// TwinCAT 3 PLC project Lab1
// ProgramVersion: 3.1.4023.0
// libraries:
//   Tc2_Standard, * (Beckhoff Automation GmbH)
//   Tc2_System, * (Beckhoff Automation GmbH)
//   Tc3_Module, * (Beckhoff Automation GmbH)
//   VisuDialogs, * (System)
// project tree:
//   DUTs/ E_CraneMode.TcDUT, E_CraneStatus.TcDUT, ST_pPistonRange.TcDUT
//   / GlobalTextList.TcGTLO, PlcTask.TcTTO (not stored), Visualization Manager.TcVMO (not stored)
//   GVLs/ HMI.TcGVL, Inputs.TcGVL, Outputs.TcGVL, Parameters.TcGVL
//   POUs/ CraneSimulation.TcPOU, F_BarToEng.TcPOU, F_LminToEng.TcPOU, F_UpdateParametersByReference.TcPOU, MAIN.TcPOU
//   VISUs/ CraneHMI.TcVIS

// ---- DUTs/E_CraneMode.TcDUT
{attribute 'qualified_only'}
{attribute 'strict'}
TYPE E_CraneMode :
(
	Manual,
	Auto
);
END_TYPE

// ---- DUTs/E_CraneStatus.TcDUT
{attribute 'qualified_only'}
{attribute 'strict'}
TYPE E_CraneStatus :
(
	Ready,
	Starting,
	Running,
	Faulty
);
END_TYPE

// ---- DUTs/ST_pPistonRange.TcDUT
TYPE ST_pPistonRange :
STRUCT
	fPistonPosMin : LREAL := 0.0;
	fPistonPosMax : LREAL := 0.5;
END_STRUCT
END_TYPE

// ---- GVLs/HMI.TcGVL
{attribute 'qualified_only'}
VAR_GLOBAL
	sPistonEndStopMessages : STRING;
END_VAR

// ---- GVLs/Inputs.TcGVL
{attribute 'qualified_only'}
VAR_GLOBAL
	bEnableSimulation : BOOL; 
	bStartSimulation : BOOL; 
	bAutoMode : BOOL; 
	fManualCylinderPositionReference : LREAL; 
	fCylinderVelocityReference : LREAL; 
END_VAR

// ---- GVLs/Outputs.TcGVL
{attribute 'qualified_only'}
VAR_GLOBAL
	fSimulationTime : LREAL; 
	bSimulationRunning : BOOL;
	fCylinderVelocity : LREAL;
	fCylinderPosition : LREAL;
	pt0_x : INT := 0;
	pt0_y : INT := 0;
	pt1_x : INT := 0;
	pt1_y : INT; 
	bPistonUpperEndStop : BOOL;
	bPistonLowerEndStop : BOOL;
END_VAR

// ---- GVLs/Parameters.TcGVL
{attribute 'qualified_only'}
VAR_GLOBAL
	fCyclicTime : LREAL := 0.01; 
	fPistonScale : LREAL :=100;	
	stPistonRange : ST_pPistonRange;
END_VAR

// ---- POUs/CraneSimulation.TcPOU
PROGRAM CraneSimulation
VAR
	fTime : LREAL; 	
	bRunning : BOOL;
	fPositionAutoMode : LREAL; 
	fInitialPosition : LREAL; 
	fInitialVelocity : LREAL;
	eStatus : E_CraneStatus;
	eMode : E_CraneMode;
	aPistonEndStopMsg : ARRAY [0..2] OF STRING := ['End Stop not active', 'Piston has reached upper End Stop', 'Piston has reached Lower End Stop'];
 	fPressureEng : REAL;
	fFlowEng : REAL;
	fPressureBar : LREAL := 60;
	fFlowLmin : LREAL := 20;
	bPistonMaxNewValue : BOOL;
	fMaxPistonPosition : LREAL;
END_VAR

IF Inputs.bStartSimulation AND Inputs.bAutoMode  THEN
	fTime := fTime + Parameters.fCyclicTime;
ELSE
	fTime := 0; 	
END_IF

IF fTime > 0 AND Inputs.bAutoMode THEN 
	bRunning := TRUE;
ELSE
	bRunning := FALSE;
END_IF

fPositionAutoMode := Inputs.fCylinderVelocityReference * 1/2*(fTime*fTime) + fInitialVelocity * fTime + fInitialPosition;

// added max/min outout value to avoid to large output for visualization
IF fPositionAutoMode >= Parameters.stPistonRange.fPistonPosMax THEN
	fPositionAutoMode := Parameters.stPistonRange.fPistonPosMax;	
ELSIF fPositionAutoMode <= Parameters.stPistonRange.fPistonPosMin  THEN
	fPositionAutoMode := Parameters.stPistonRange.fPistonPosMin; 
ELSE	
	fPositionAutoMode := fPositionAutoMode;
END_IF

IF Inputs.bAutoMode THEN
	Outputs.fCylinderPosition := fPositionAutoMode;
ELSE
	Outputs.fCylinderPosition := Inputs.fManualCylinderPositionReference;	
END_IF


Outputs.bSimulationRunning := bRunning;  
Outputs.fSimulationTime := fTime; 
Outputs.fCylinderVelocity := Inputs.fCylinderVelocityReference;
Outputs.pt1_y := LREAL_TO_INT(Outputs.fCylinderPosition * Parameters.fPistonScale);

//status
IF inputs.bEnableSimulation THEN
	eStatus := E_CraneStatus.Ready;
ELSE
	eStatus := E_CraneStatus.Faulty;
END_IF

IF inputs.bStartSimulation THEN
	eStatus := E_CraneStatus.Starting;
END_IF

IF Outputs.bSimulationRunning THEN
	eStatus := E_CraneStatus.Running;
END_IF

//mode
IF inputs.bAutoMode THEN
	eMode := E_CraneMode.Auto;
ELSE
	eMode := E_CraneMode.Manual;
END_IF

//Logic for pistonStops
IF Outputs.fCylinderPosition <= Parameters.stPistonRange.fPistonPosMin THEN
	Outputs.bPistonLowerEndStop := TRUE;
	Outputs.bPistonUpperEndStop := FALSE;
	HMI.sPistonEndStopMessages := aPistonEndStopMsg[2];
	
ELSIF Outputs.fCylinderPosition >= Parameters.stPistonRange.fPistonPosMax THEN
	Outputs.bPistonLowerEndStop := FALSE;
	Outputs.bPistonUpperEndStop := TRUE;
	HMI.sPistonEndStopMessages := aPistonEndStopMsg[1];

ELSE
	Outputs.bPistonLowerEndStop := FALSE;
	Outputs.bPistonUpperEndStop := FALSE;
	HMI.sPistonEndStopMessages := aPistonEndStopMsg[0];
END_IF

//unit conversions

fPressureEng := LREAL_TO_REAL (F_BarToEng(fBar := fPressureBar));
fFlowEng := LREAL_TO_REAL (F_LminToEng(fLminFlow := fFlowLmin));

//Piston stroke

F_UpdateParametersByReference(
	bSetNewValue := bPistonMaxNewValue,
	fMaxPistonStroke := fMaxPistonPosition,
	paramCylinderPiston := Parameters.stPistonRange
);

END_PROGRAM

// ---- POUs/F_BarToEng.TcPOU
FUNCTION F_BarToEng : LREAL
VAR_INPUT
	fBar : LREAL;
	
END_VAR
VAR
END_VAR

F_BarToEng := fBar*1E5;

END_FUNCTION

// ---- POUs/F_LminToEng.TcPOU
FUNCTION F_LminToEng : LREAL
VAR_INPUT
	fLminFlow : LREAL;
END_VAR
VAR
END_VAR

F_LminToEng := fLminFlow / 60000;

END_FUNCTION

// ---- POUs/F_UpdateParametersByReference.TcPOU
FUNCTION F_UpdateParametersByReference
VAR_INPUT
	bSetNewValue : BOOL;
	fMaxPistonStroke : LREAL;
	paramCylinderPiston : REFERENCE TO ST_pPistonRange;
END_VAR
VAR
END_VAR

IF bSetNewValue THEN
	paramCylinderPiston.fPistonPosMax := fMaxPistonStroke;
	bSetNewValue := FALSE;
END_IF

END_FUNCTION

// ---- POUs/MAIN.TcPOU
PROGRAM MAIN
VAR
END_VAR

CraneSimulation();

END_PROGRAM

// ---- GlobalTextList.TcGTLO
TEXTLIST GlobalTextList
  624 = '%0.1f'
  198 = '%f'
  949 = '%i'
  819 = '%s'
  175 = 'AUTO'
  236 = 'Clock: %s [s]'
  226 = 'Current Max Range: %f'
  957 = 'Current Max: %f'
  995 = 'Cylinder Position Reference: %f [m]'
  752 = 'Cylinder Velocity Reference: %0.0001f [m/s]'
  954 = 'Cylinder Velocity Reference: %0.01f [m/s]'
  105 = 'Cylinder Velocity Reference: %0.1f [m/s]'
  755 = 'Cylinder Velocity Reference: %0.1s [m/s]'
  25 = 'Cylinder Velocity Reference: %f [m/s]'
  308 = 'Cylinder Velocity Reference: %f [m]'
  30 = 'Cylinder Velocity Reference: %i'
  903 = 'Cylinder Velocity Reference: %s'
  128 = 'Cylinder Velocity Reference: %s [m/s]'
  353 = 'Enable'
  409 = 'ENABLE'
  796 = 'Enter new max position'
  744 = 'Enter new max position: %f'
  660 = 'MANUAL'
  8 = 'Manual Cylinder Position   Reference [m]'
  157 = 'Manual Cylinder Position Reference'
  935 = 'Mode: %s'
  310 = 'RUNNING'
  808 = 'Set new max position'
  466 = 'Simulation'
  279 = 'Start'
  868 = 'START'
  978 = 'Started'
  645 = 'Status: %s'
  495 = 'Time: %0.1f [s]'
  221 = 'Time: %f [s]'
  61 = 'Time: %i [s]'
  725 = 'Time: %s [s]'
  444 = 'x0'
END_TEXTLIST

// ---- VISUs/CraneHMI.TcVIS
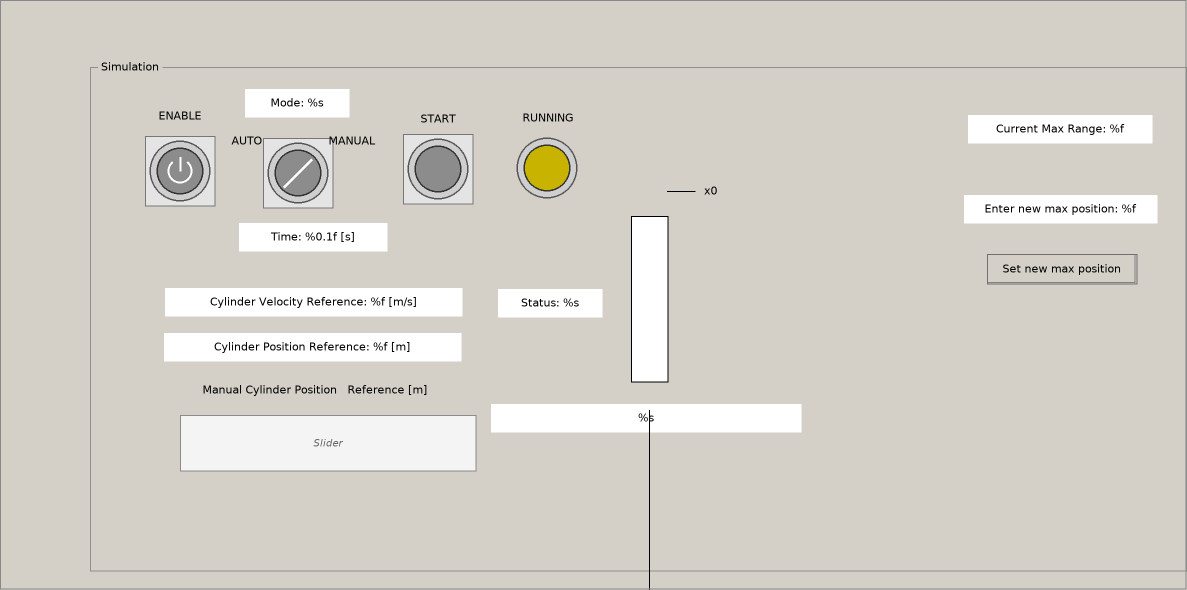
VISUALIZATION CraneHMI  // 1187x590
    Rectangle (566,281 166x37), angle 270
    GroupBox (90,59 1097x512), "Simulation"
        PowerSwitch (55,77 70x70), variable: Inputs.bEnableSimulation, behaviour: TOGGLE, style: Switch-PowerSwitch-Gray
        PushSwitch (313,75 70x70), variable: Inputs.bStartSimulation, behaviour: TOGGLE, style: Switch-PushSwitch-Gray
        Lamp1 (422,74 70x70), variable: Outputs.bSimulationRunning, style: Lamp-Lamp1-Yellow
        Textfield (74,228 299x30), "Cylinder Velocity Reference: %f [m/s]", text variable: Inputs.fCylinderVelocityReference
            OnMouseClick: write the text variable via Default
        Label (15,42 150x30), "ENABLE"
        Label (273,45 150x30), "START"
        Label (383,44 150x30), "RUNNING"
        Textfield (148,163 150x30), "Time: %0.1f [s]", text variable: Outputs.fSimulationTime
        Slider (90,356 296x56), variable: Inputs.fManualCylinderPositionReference, scale 0..1
        RotarySwitch (173,79 70x70), variable: Inputs.bAutoMode, behaviour: TOGGLE, style: Switch-RotarySwitch-Gray
        Label (82,67 150x30), "AUTO"
        Label (187,67 150x30), "MANUAL"
        Label (90,316 270x30), "Manual Cylinder Position Reference [m]"
        Textfield (73,273 299x30), "Cylinder Position Reference: %f [m]", text variable: Inputs.fManualCylinderPositionReference
        Line (577,132) (605,132)
        Label (607,117 28x30), "x0"
        Textfield (407,229 106x30), "Status: %s", text variable: CraneSimulation.eStatus
        Textfield (154,29 106x30), "Mode: %s", text variable: CraneSimulation.eMode
        Textfield (400,344 312x30), "%s", text variable: HMI.sPistonEndStopMessages
        Textfield (877,55 186x30), "Current Max Range: %f", text variable: Parameters.stPistonRange.fPistonPosMax
        Textfield (873,135 195x30), "Enter new max position: %f", text variable: CraneSimulation.fMaxPistonPosition
            OnMouseDown: write the text variable via Default, min 0, max 0.5
        Button (897,195 150x30), "Set new max position"
            tap CraneSimulation.bPistonMaxNewValue
    Line (649,410) (649,590)
        p1126004900: Outputs.pt1_y
        p3528305787: Outputs.pt0_x
        p2773130477: Outputs.pt0_y
        p874137650: Outputs.pt1_x
    Line (706,188) (706,188)
END_VISUALIZATION
